PROGRAM MAIN
VAR
END_VAR

MAIN_LIB_Python();

END_PROGRAM

(* stored: Version 1.1.0.1, ProductVersion 3.1.4024.12
   POU MAIN: Id {04f9be17-5a8d-423f-ad43-2a1ef120b01d}, SpecialFunc None *)
